// TwinCAT 3 PLC project Cluster_Controller
// ProgramVersion: 3.1.4022.7
// libraries:
//   Tc2_Standard, * (Beckhoff Automation GmbH)
//   Tc2_System, * (Beckhoff Automation GmbH)
//   Tc3_Module, * (Beckhoff Automation GmbH)
// project tree:
//   GVLs/ GVL_CONVERTER.TcGVL
//   / PlcTask.TcTTO
//   POUs/ MAIN.TcPOU
// real-time tasks:
//   TASK PlcTask: cycle T#10ms, priority 20, ADS port 350

CONFIGURATION Cluster_Controller
    RESOURCE PLC ON TwinCAT3
        TASK PlcTask(INTERVAL := T#10ms, PRIORITY := 20);
        PROGRAM MAIN WITH PlcTask : MAIN;
    END_RESOURCE
END_CONFIGURATION

// ---- GVLs/GVL_CONVERTER.TcGVL
{attribute 'qualified_only'}
VAR_GLOBAL
	uiStateCmd:UINT;
END_VAR

// ---- POUs/MAIN.TcPOU
PROGRAM MAIN
VAR
END_VAR

END_PROGRAM
